// TIA Portal V20 export
FUNCTION_BLOCK "LER_Thickness"   // FB10, LAD
// stored: Access Published, MemoryReserve 100, SetENOAutomatically false
   VAR_INPUT
      enable : Bool := true;
      enableManualCmds : Bool;
      productUnused : Bool;   // Unused is simulation, dryrun etc..
      errAckHmi : Bool;
   END_VAR
   VAR_OUTPUT
      error : Bool;
      errorCode : Word;
   END_VAR
   VAR_IN_OUT
      configuration : "LER_typeThicknessConfiguration";
      moduleInterface : "LER_typeThicknessInterface";
      controlNodes : "LER_typeThicknessControlNode";
   END_VAR
   VAR
      statLVDTCmd { S7_SetPoint := 'True'} : "LER_typeThicknessCommand";
      statLVDTProfinetInput { S7_SetPoint := 'True'} : "LER_typeThicknessProfinetInput";
      statLVDTProfinetOutput { S7_SetPoint := 'True'} : "LER_typeThicknessProfinetOutput";
      statMonitoring : "LER_typeThicknessMonitoring";
      statLvdtConfig { S7_SetPoint := 'True'} : "LER_typeThicknessConfiguration";
      statRetValInt : Array[1..#count] of Int;
      statRetValWord { ExternalAccessible := 'False'; ExternalVisible := 'False'; ExternalWritable := 'False'} : Array[1..#count] of Word;
      instTON { S7_SetPoint := 'True'} : Array[0..4] of TON_TIME;
      statBit { S7_SetPoint := 'True'} : Array[0..49] of Bool;
      statRowDataDint_always : Array[0..3] of DInt;
      statRowDataReal_always : Array[0..3] of Real;
      statRowDataDint_capture : Array[0..3] of DInt;
      statRowDataReal_capture : Array[0..3] of Real;
      statTonTimer { S7_SetPoint := 'True'} : Array[0..99] of TON_TIME;
      statPulse { S7_SetPoint := 'True'} : Array[0..99] of Bool;
   END_VAR
   VAR_TEMP
      tempRetVal : Array[1..#count] of Int;
      tempIndex : Int;
   END_VAR
   VAR CONSTANT
      delayTime : Time := T#2s;
      count : Int := 10;
      scaleData : DInt := 256;
      scaleDigit : Real := 10000.0;
      statusNoErrorOccurred : Word := 16#0000;   // No error occurred.
      ioDeviceError : Word := 16#8000;
      ampError : Word := 16#8002;
      errHwdNotConfigured : Word := 16#8090;   // You have not configured a module for the specified hardware identifier or You have ignored the restriction concerning the length of consistent data, or you have not specified a hardware identifier as an address at parameter LADDR
      errRecordDataType : Word := 16#8092;   // Non-supported data type in the RECORD parameter.
      errNoDpProfinetIoModule : Word := 16#8093;   // No DP module/PROFINET IO device from which you can read consistent data exists for the hardware identifier specified in LADDR . This error code also occurs if the module addressed by means of LADDR does not have inputs.
      errIoAccessPermission : Word := 16#80A0;   // An access error was detected when accessing the I/O.
      errRecordLengthInsufficient : Word := 16#80B1;   // The length of the specified destination area at parameter RECORD is shorter than the configured user data length.
      errDataNotReceived : Word := 16#80C0;   // The data have not been read yet.
   END_VAR
   // // statBit[20] : amp0 OK
   // // statBit[21] : amp1 OK
   // // statBit[22] : amp2 OK
   // // statBit[23] : amp3 OK
   // // statBit[25] : Total OK
   // // statBit[30] : amp0 NG
   // // statBit[31] : amp1 NG
   // // statBit[32] : amp2 NG
   // // statBit[33] : amp3 NG
   // // statBit[35] : One or more NG
   // // statBit[40] : Busy
   // // statBit[41] : Complete
   // // statBit[45] : P_TRIG
   VAR_TEMP   // added for the SCL form of the ladder/FBD networks
      _w1 : Bool;
      _w2 : Bool;
      _w3 : Bool;
      _w4 : Bool;
      _w5 : Bool;
   END_VAR
BEGIN

REGION Network 1 (SCL): DP READ
   REGION DP read

       IF #enable AND NOT #productUnused THEN
           #statRetValInt[1] := DPRD_DAT(LADDR := #configuration.hwID.interfaceControllerID, RECORD => #statLVDTProfinetInput.interfaceController);
           #statRetValInt[2] := DPRD_DAT(LADDR := #configuration.hwID.ampID[0], RECORD => #statLVDTProfinetInput.amp[0]);
           #statRetValInt[3] := DPRD_DAT(LADDR := #configuration.hwID.ampID[1], RECORD => #statLVDTProfinetInput.amp[1]);
           #statRetValInt[4] := DPRD_DAT(LADDR := #configuration.hwID.ampID[2], RECORD => #statLVDTProfinetInput.amp[2]);
           #statRetValInt[5] := DPRD_DAT(LADDR := #configuration.hwID.ampID[3], RECORD => #statLVDTProfinetInput.amp[3]);
       END_IF;

   END_REGION
END_REGION

REGION Network 2 (SCL): INPUT MAPPING
   REGION Input mapping

       IF #enable THEN
           IF #enableManualCmds THEN
               #statLVDTCmd := #moduleInterface.command;
               #statLvdtConfig := #moduleInterface.configuration;
           ELSE
               #statLVDTCmd := #controlNodes.command;
               #statLvdtConfig := #configuration;
           END_IF;
       END_IF;

   END_REGION
END_REGION

REGION Network 3 (SCL): ERROR STATUS
   REGION Error check

       IF #enable AND NOT #productUnused THEN
           IF #statRetValInt <> #tempRetVal THEN
               FOR #tempIndex := 1 TO #count DO
                   #statRetValWord[#tempIndex] := INT_TO_WORD(#statRetValInt[#tempIndex]);
                   CASE #statRetValWord[#tempIndex] OF

                       #errHwdNotConfigured:
                           #errorCode := #errHwdNotConfigured;

                       #errRecordDataType:
                           #errorCode := #errRecordDataType;

                       #errNoDpProfinetIoModule:
                           #errorCode := #errNoDpProfinetIoModule;

                       #errIoAccessPermission:
                           #errorCode := #errIoAccessPermission;

                       #errRecordLengthInsufficient:
                           #errorCode := #errRecordLengthInsufficient;

                       #errDataNotReceived:
                           #errorCode := #errDataNotReceived;
                   END_CASE;
               END_FOR;

           ELSIF #statLVDTProfinetInput.interfaceController.b07ErrorStatus THEN
               #errorCode := #ioDeviceError;

           ELSIF #statLVDTProfinetInput.amp[0].b17ErrorStatus OR
               #statLVDTProfinetInput.amp[1].b17ErrorStatus OR
               #statLVDTProfinetInput.amp[2].b17ErrorStatus OR
               #statLVDTProfinetInput.amp[3].b17ErrorStatus THEN
               #errorCode := #ampError;

           ELSE
               #errorCode := #statusNoErrorOccurred;
           END_IF;
       ELSE
           #errorCode := #statusNoErrorOccurred;
       END_IF;

       #error := #errorCode <> 0;

   END_REGION
END_REGION

REGION Network 4: SEQUENCE : READY
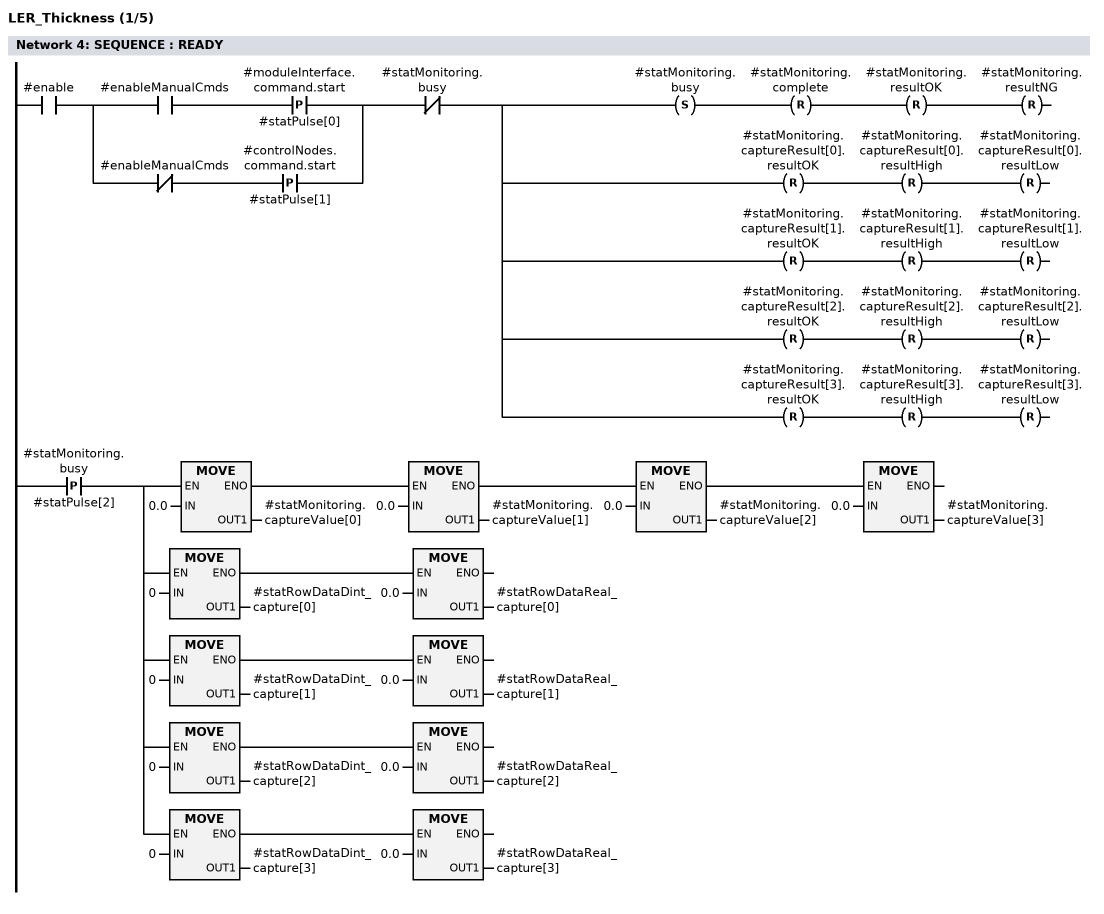
   RUNG wire#powerrail
      Contact( #enable )
      wire#w1
      Contact( #enableManualCmds )
      P_Contact(operand := #moduleInterface.command.start, bit := #statPulse[0])
      wire#w2
      I_Contact( #statMonitoring.busy )
      wire#w3
      S_Coil( #statMonitoring.busy )
      R_Coil( #statMonitoring.complete )
      R_Coil( #statMonitoring.resultOK )
      R_Coil( #statMonitoring.resultNG )
   END_RUNG
   RUNG wire#w1
      I_Contact( #enableManualCmds )
      P_Contact(operand := #controlNodes.command.start, bit := #statPulse[1])
   END_RUNG wire#w2
   RUNG wire#w3
      R_Coil( #statMonitoring.captureResult[0].resultOK )
      R_Coil( #statMonitoring.captureResult[0].resultHigh )
      R_Coil( #statMonitoring.captureResult[0].resultLow )
   END_RUNG
   RUNG wire#w3
      R_Coil( #statMonitoring.captureResult[1].resultOK )
      R_Coil( #statMonitoring.captureResult[1].resultHigh )
      R_Coil( #statMonitoring.captureResult[1].resultLow )
   END_RUNG
   RUNG wire#w3
      R_Coil( #statMonitoring.captureResult[2].resultOK )
      R_Coil( #statMonitoring.captureResult[2].resultHigh )
      R_Coil( #statMonitoring.captureResult[2].resultLow )
   END_RUNG
   RUNG wire#w3
      R_Coil( #statMonitoring.captureResult[3].resultOK )
      R_Coil( #statMonitoring.captureResult[3].resultHigh )
      R_Coil( #statMonitoring.captureResult[3].resultLow )
   END_RUNG
   RUNG wire#powerrail
      P_Contact(operand := #statMonitoring.busy, bit := #statPulse[2])
      wire#w4
      Move(in := 0.0, out1 => #statMonitoring.captureValue[0])
      Move(in := 0.0, out1 => #statMonitoring.captureValue[1])
      Move(in := 0.0, out1 => #statMonitoring.captureValue[2])
      Move(in := 0.0, out1 => #statMonitoring.captureValue[3])
   END_RUNG
   RUNG wire#w4
      Move(in := 0, out1 => #statRowDataDint_capture[0])
      Move(in := 0.0, out1 => #statRowDataReal_capture[0])
   END_RUNG
   RUNG wire#w4
      Move(in := 0, out1 => #statRowDataDint_capture[1])
      Move(in := 0.0, out1 => #statRowDataReal_capture[1])
   END_RUNG
   RUNG wire#w4
      Move(in := 0, out1 => #statRowDataDint_capture[2])
      Move(in := 0.0, out1 => #statRowDataReal_capture[2])
   END_RUNG
   RUNG wire#w4
      Move(in := 0, out1 => #statRowDataDint_capture[3])
      Move(in := 0.0, out1 => #statRowDataReal_capture[3])
   END_RUNG
   // the same network as SCL:
   #_w1 := #enable AND #enableManualCmds AND #moduleInterface.command.start AND NOT #statPulse[0];   // rising edge of #moduleInterface.command.start
   #statPulse[0] := #moduleInterface.command.start;
   #_w2 := #enable AND NOT #enableManualCmds AND #controlNodes.command.start AND NOT #statPulse[1];   // rising edge of #controlNodes.command.start
   #statPulse[1] := #controlNodes.command.start;
   #_w3 := (#_w1 OR #_w2) AND NOT #statMonitoring.busy;
   IF #_w3 THEN
       #statMonitoring.busy := TRUE;
       #statMonitoring.complete := FALSE;
       #statMonitoring.resultOK := FALSE;
       #statMonitoring.resultNG := FALSE;
       #statMonitoring.captureResult[0].resultOK := FALSE;
       #statMonitoring.captureResult[0].resultHigh := FALSE;
       #statMonitoring.captureResult[0].resultLow := FALSE;
       #statMonitoring.captureResult[1].resultOK := FALSE;
       #statMonitoring.captureResult[1].resultHigh := FALSE;
       #statMonitoring.captureResult[1].resultLow := FALSE;
       #statMonitoring.captureResult[2].resultOK := FALSE;
       #statMonitoring.captureResult[2].resultHigh := FALSE;
       #statMonitoring.captureResult[2].resultLow := FALSE;
       #statMonitoring.captureResult[3].resultOK := FALSE;
       #statMonitoring.captureResult[3].resultHigh := FALSE;
       #statMonitoring.captureResult[3].resultLow := FALSE;
   END_IF;
   #_w4 := #statMonitoring.busy AND NOT #statPulse[2];   // rising edge of #statMonitoring.busy
   #statPulse[2] := #statMonitoring.busy;
   IF #_w4 THEN
       #statMonitoring.captureValue[0] := 0.0;
       #statMonitoring.captureValue[1] := 0.0;
       #statMonitoring.captureValue[2] := 0.0;
       #statMonitoring.captureValue[3] := 0.0;
       #statRowDataDint_capture[0] := 0;
       #statRowDataReal_capture[0] := 0.0;
       #statRowDataDint_capture[1] := 0;
       #statRowDataReal_capture[1] := 0.0;
       #statRowDataDint_capture[2] := 0;
       #statRowDataReal_capture[2] := 0.0;
       #statRowDataDint_capture[3] := 0;
       #statRowDataReal_capture[3] := 0.0;
   END_IF;
END_REGION

REGION Network 5: SEQUENCE : START
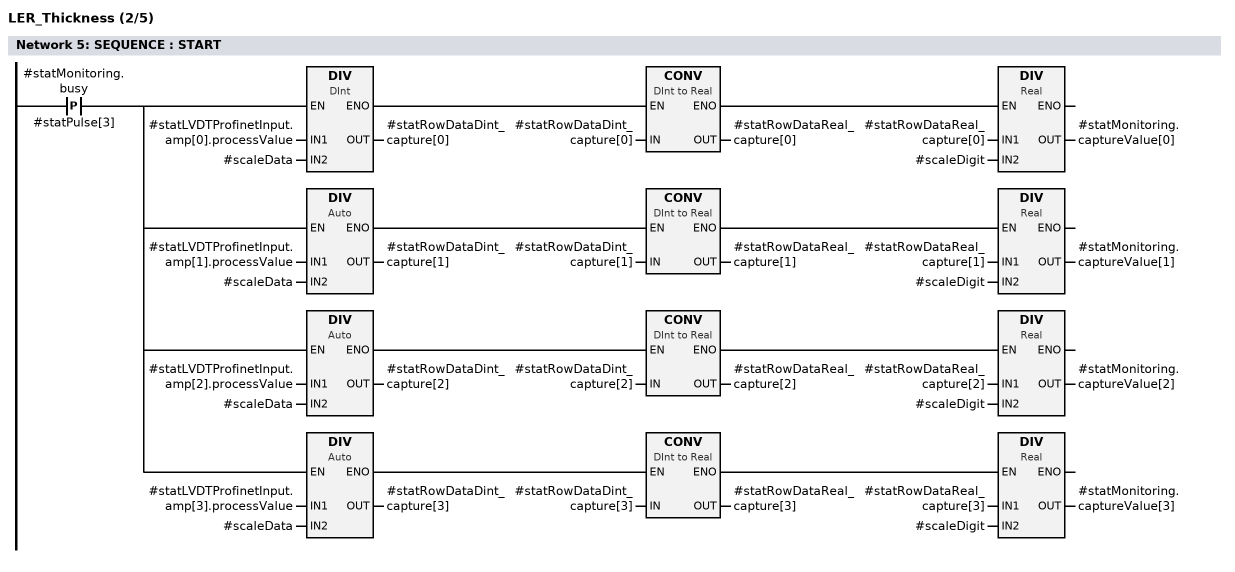
   RUNG wire#powerrail
      P_Contact(operand := #statMonitoring.busy, bit := #statPulse[3])
      wire#w1
      { S7_Templates := "SrcType := DInt" } Div(in1 := #statLVDTProfinetInput.amp[0].processValue, in2 := #scaleData, out => #statRowDataDint_capture[0])
      { S7_Templates := "[SrcType := DInt, DestType := Real]" } Convert(in := #statRowDataDint_capture[0], out => #statRowDataReal_capture[0])
      { S7_Templates := "SrcType := Real" } Div(in1 := #statRowDataReal_capture[0], in2 := #scaleDigit, out => #statMonitoring.captureValue[0])
   END_RUNG
   RUNG wire#w1
      Div(in1 := #statLVDTProfinetInput.amp[1].processValue, in2 := #scaleData, out => #statRowDataDint_capture[1])
      { S7_Templates := "[SrcType := DInt, DestType := Real]" } Convert(in := #statRowDataDint_capture[1], out => #statRowDataReal_capture[1])
      { S7_Templates := "SrcType := Real" } Div(in1 := #statRowDataReal_capture[1], in2 := #scaleDigit, out => #statMonitoring.captureValue[1])
   END_RUNG
   RUNG wire#w1
      Div(in1 := #statLVDTProfinetInput.amp[2].processValue, in2 := #scaleData, out => #statRowDataDint_capture[2])
      { S7_Templates := "[SrcType := DInt, DestType := Real]" } Convert(in := #statRowDataDint_capture[2], out => #statRowDataReal_capture[2])
      { S7_Templates := "SrcType := Real" } Div(in1 := #statRowDataReal_capture[2], in2 := #scaleDigit, out => #statMonitoring.captureValue[2])
   END_RUNG
   RUNG wire#w1
      Div(in1 := #statLVDTProfinetInput.amp[3].processValue, in2 := #scaleData, out => #statRowDataDint_capture[3])
      { S7_Templates := "[SrcType := DInt, DestType := Real]" } Convert(in := #statRowDataDint_capture[3], out => #statRowDataReal_capture[3])
      { S7_Templates := "SrcType := Real" } Div(in1 := #statRowDataReal_capture[3], in2 := #scaleDigit, out => #statMonitoring.captureValue[3])
   END_RUNG
   // the same network as SCL:
   #_w1 := #statMonitoring.busy AND NOT #statPulse[3];   // rising edge of #statMonitoring.busy
   #statPulse[3] := #statMonitoring.busy;
   IF #_w1 THEN
       #statRowDataDint_capture[0] := #statLVDTProfinetInput.amp[0].processValue / #scaleData;
       #statRowDataReal_capture[0] := DINT_TO_REAL(#statRowDataDint_capture[0]);
       #statMonitoring.captureValue[0] := #statRowDataReal_capture[0] / #scaleDigit;
       #statRowDataDint_capture[1] := #statLVDTProfinetInput.amp[1].processValue / #scaleData;
       #statRowDataReal_capture[1] := DINT_TO_REAL(#statRowDataDint_capture[1]);
       #statMonitoring.captureValue[1] := #statRowDataReal_capture[1] / #scaleDigit;
       #statRowDataDint_capture[2] := #statLVDTProfinetInput.amp[2].processValue / #scaleData;
       #statRowDataReal_capture[2] := DINT_TO_REAL(#statRowDataDint_capture[2]);
       #statMonitoring.captureValue[2] := #statRowDataReal_capture[2] / #scaleDigit;
       #statRowDataDint_capture[3] := #statLVDTProfinetInput.amp[3].processValue / #scaleData;
       #statRowDataReal_capture[3] := DINT_TO_REAL(#statRowDataDint_capture[3]);
       #statMonitoring.captureValue[3] := #statRowDataReal_capture[3] / #scaleDigit;
   END_IF;
END_REGION

REGION Network 6: SEQUENCE : RESULT
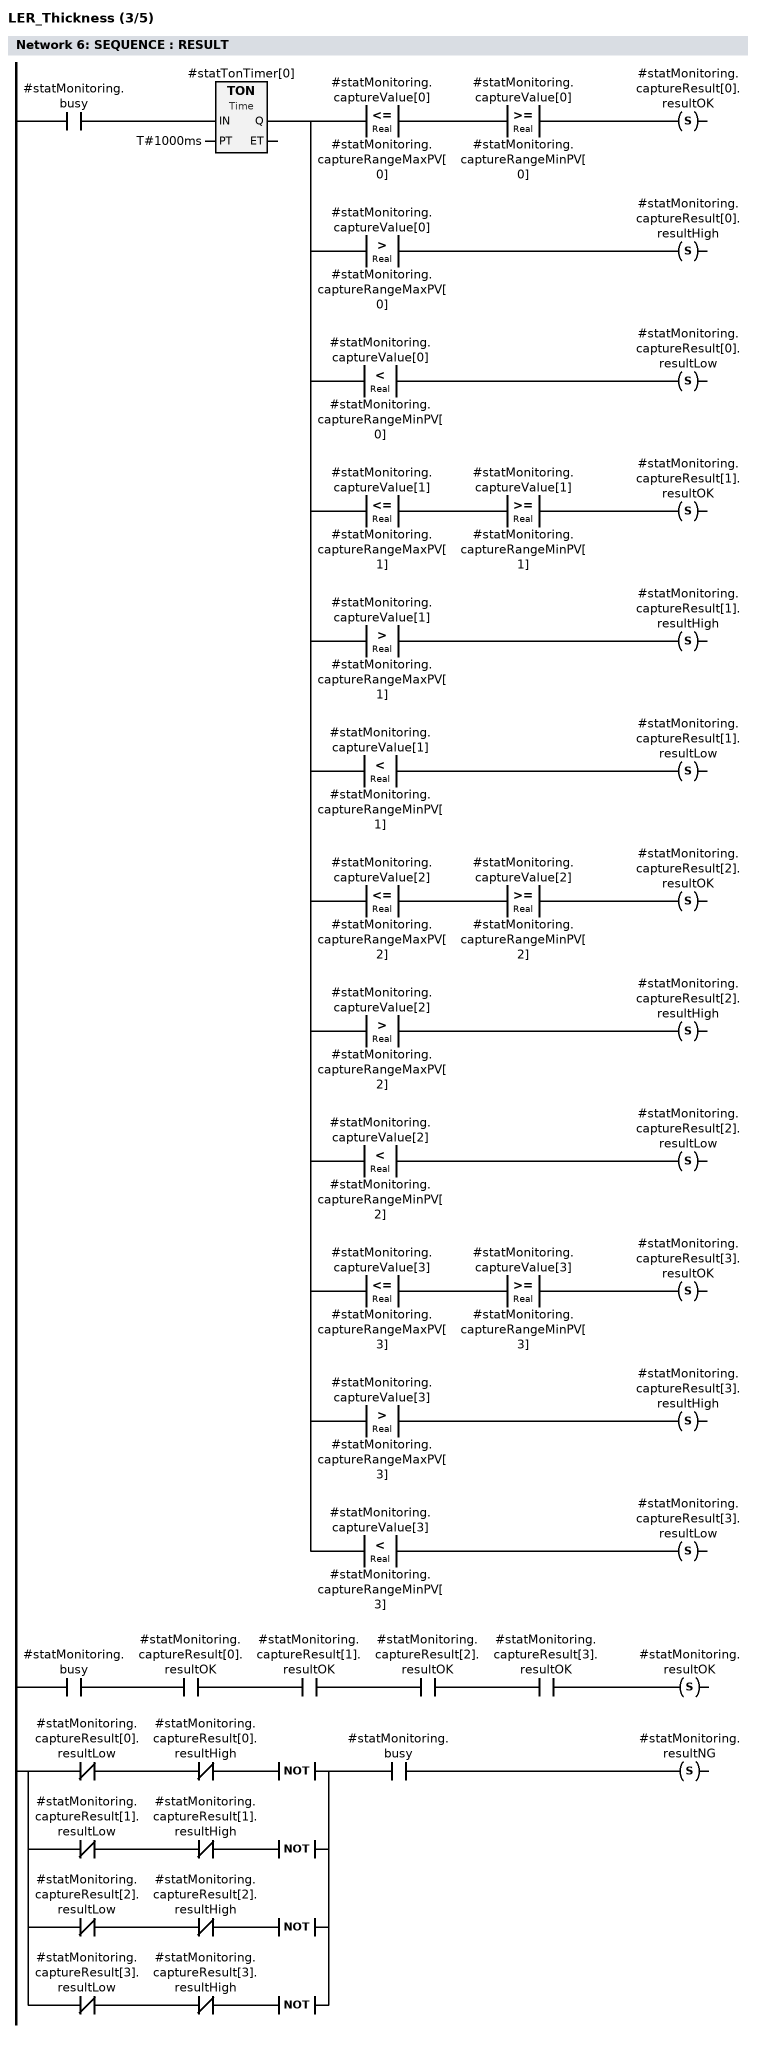
   RUNG wire#powerrail
      Contact( #statMonitoring.busy )
      { S7_Templates := "time_type := Time" } #statTonTimer[0].TON(pt := T#1000ms, et =>)
      wire#w1
      { S7_Templates := "SrcType := Real" } LE_Contact(in1 := #statMonitoring.captureValue[0], in2 := #statMonitoring.captureRangeMaxPV[0])
      { S7_Templates := "SrcType := Real" } GE_Contact(in1 := #statMonitoring.captureValue[0], in2 := #statMonitoring.captureRangeMinPV[0])
      S_Coil( #statMonitoring.captureResult[0].resultOK )
   END_RUNG
   RUNG wire#w1
      { S7_Templates := "SrcType := Real" } GT_Contact(in1 := #statMonitoring.captureValue[0], in2 := #statMonitoring.captureRangeMaxPV[0])
      S_Coil( #statMonitoring.captureResult[0].resultHigh )
   END_RUNG
   RUNG wire#w1
      { S7_Templates := "SrcType := Real" } LT_Contact(in1 := #statMonitoring.captureValue[0], in2 := #statMonitoring.captureRangeMinPV[0])
      S_Coil( #statMonitoring.captureResult[0].resultLow )
   END_RUNG
   RUNG wire#w1
      { S7_Templates := "SrcType := Real" } LE_Contact(in1 := #statMonitoring.captureValue[1], in2 := #statMonitoring.captureRangeMaxPV[1])
      { S7_Templates := "SrcType := Real" } GE_Contact(in1 := #statMonitoring.captureValue[1], in2 := #statMonitoring.captureRangeMinPV[1])
      S_Coil( #statMonitoring.captureResult[1].resultOK )
   END_RUNG
   RUNG wire#w1
      { S7_Templates := "SrcType := Real" } GT_Contact(in1 := #statMonitoring.captureValue[1], in2 := #statMonitoring.captureRangeMaxPV[1])
      S_Coil( #statMonitoring.captureResult[1].resultHigh )
   END_RUNG
   RUNG wire#w1
      { S7_Templates := "SrcType := Real" } LT_Contact(in1 := #statMonitoring.captureValue[1], in2 := #statMonitoring.captureRangeMinPV[1])
      S_Coil( #statMonitoring.captureResult[1].resultLow )
   END_RUNG
   RUNG wire#w1
      { S7_Templates := "SrcType := Real" } LE_Contact(in1 := #statMonitoring.captureValue[2], in2 := #statMonitoring.captureRangeMaxPV[2])
      { S7_Templates := "SrcType := Real" } GE_Contact(in1 := #statMonitoring.captureValue[2], in2 := #statMonitoring.captureRangeMinPV[2])
      S_Coil( #statMonitoring.captureResult[2].resultOK )
   END_RUNG
   RUNG wire#w1
      { S7_Templates := "SrcType := Real" } GT_Contact(in1 := #statMonitoring.captureValue[2], in2 := #statMonitoring.captureRangeMaxPV[2])
      S_Coil( #statMonitoring.captureResult[2].resultHigh )
   END_RUNG
   RUNG wire#w1
      { S7_Templates := "SrcType := Real" } LT_Contact(in1 := #statMonitoring.captureValue[2], in2 := #statMonitoring.captureRangeMinPV[2])
      S_Coil( #statMonitoring.captureResult[2].resultLow )
   END_RUNG
   RUNG wire#w1
      { S7_Templates := "SrcType := Real" } LE_Contact(in1 := #statMonitoring.captureValue[3], in2 := #statMonitoring.captureRangeMaxPV[3])
      { S7_Templates := "SrcType := Real" } GE_Contact(in1 := #statMonitoring.captureValue[3], in2 := #statMonitoring.captureRangeMinPV[3])
      S_Coil( #statMonitoring.captureResult[3].resultOK )
   END_RUNG
   RUNG wire#w1
      { S7_Templates := "SrcType := Real" } GT_Contact(in1 := #statMonitoring.captureValue[3], in2 := #statMonitoring.captureRangeMaxPV[3])
      S_Coil( #statMonitoring.captureResult[3].resultHigh )
   END_RUNG
   RUNG wire#w1
      { S7_Templates := "SrcType := Real" } LT_Contact(in1 := #statMonitoring.captureValue[3], in2 := #statMonitoring.captureRangeMinPV[3])
      S_Coil( #statMonitoring.captureResult[3].resultLow )
   END_RUNG
   RUNG wire#powerrail
      Contact( #statMonitoring.busy )
      Contact( #statMonitoring.captureResult[0].resultOK )
      Contact( #statMonitoring.captureResult[1].resultOK )
      Contact( #statMonitoring.captureResult[2].resultOK )
      Contact( #statMonitoring.captureResult[3].resultOK )
      S_Coil( #statMonitoring.resultOK )
   END_RUNG
   RUNG wire#powerrail
      I_Contact( #statMonitoring.captureResult[0].resultLow )
      I_Contact( #statMonitoring.captureResult[0].resultHigh )
      Not()
      wire#w2
      Contact( #statMonitoring.busy )
      S_Coil( #statMonitoring.resultNG )
   END_RUNG
   RUNG wire#powerrail
      I_Contact( #statMonitoring.captureResult[1].resultLow )
      I_Contact( #statMonitoring.captureResult[1].resultHigh )
      Not()
   END_RUNG wire#w2
   RUNG wire#powerrail
      I_Contact( #statMonitoring.captureResult[2].resultLow )
      I_Contact( #statMonitoring.captureResult[2].resultHigh )
      Not()
   END_RUNG wire#w2
   RUNG wire#powerrail
      I_Contact( #statMonitoring.captureResult[3].resultLow )
      I_Contact( #statMonitoring.captureResult[3].resultHigh )
      Not()
   END_RUNG wire#w2
   // the same network as SCL:
   #statTonTimer[0].TON(IN := #statMonitoring.busy, PT := T#1000ms);
   IF #statTonTimer[0].Q AND (#statMonitoring.captureValue[0] <= #statMonitoring.captureRangeMaxPV[0]) AND (#statMonitoring.captureValue[0] >= #statMonitoring.captureRangeMinPV[0]) THEN
       #statMonitoring.captureResult[0].resultOK := TRUE;
   END_IF;
   IF #statTonTimer[0].Q AND (#statMonitoring.captureValue[0] > #statMonitoring.captureRangeMaxPV[0]) THEN
       #statMonitoring.captureResult[0].resultHigh := TRUE;
   END_IF;
   IF #statTonTimer[0].Q AND (#statMonitoring.captureValue[0] < #statMonitoring.captureRangeMinPV[0]) THEN
       #statMonitoring.captureResult[0].resultLow := TRUE;
   END_IF;
   IF #statTonTimer[0].Q AND (#statMonitoring.captureValue[1] <= #statMonitoring.captureRangeMaxPV[1]) AND (#statMonitoring.captureValue[1] >= #statMonitoring.captureRangeMinPV[1]) THEN
       #statMonitoring.captureResult[1].resultOK := TRUE;
   END_IF;
   IF #statTonTimer[0].Q AND (#statMonitoring.captureValue[1] > #statMonitoring.captureRangeMaxPV[1]) THEN
       #statMonitoring.captureResult[1].resultHigh := TRUE;
   END_IF;
   IF #statTonTimer[0].Q AND (#statMonitoring.captureValue[1] < #statMonitoring.captureRangeMinPV[1]) THEN
       #statMonitoring.captureResult[1].resultLow := TRUE;
   END_IF;
   IF #statTonTimer[0].Q AND (#statMonitoring.captureValue[2] <= #statMonitoring.captureRangeMaxPV[2]) AND (#statMonitoring.captureValue[2] >= #statMonitoring.captureRangeMinPV[2]) THEN
       #statMonitoring.captureResult[2].resultOK := TRUE;
   END_IF;
   IF #statTonTimer[0].Q AND (#statMonitoring.captureValue[2] > #statMonitoring.captureRangeMaxPV[2]) THEN
       #statMonitoring.captureResult[2].resultHigh := TRUE;
   END_IF;
   IF #statTonTimer[0].Q AND (#statMonitoring.captureValue[2] < #statMonitoring.captureRangeMinPV[2]) THEN
       #statMonitoring.captureResult[2].resultLow := TRUE;
   END_IF;
   IF #statTonTimer[0].Q AND (#statMonitoring.captureValue[3] <= #statMonitoring.captureRangeMaxPV[3]) AND (#statMonitoring.captureValue[3] >= #statMonitoring.captureRangeMinPV[3]) THEN
       #statMonitoring.captureResult[3].resultOK := TRUE;
   END_IF;
   IF #statTonTimer[0].Q AND (#statMonitoring.captureValue[3] > #statMonitoring.captureRangeMaxPV[3]) THEN
       #statMonitoring.captureResult[3].resultHigh := TRUE;
   END_IF;
   IF #statTonTimer[0].Q AND (#statMonitoring.captureValue[3] < #statMonitoring.captureRangeMinPV[3]) THEN
       #statMonitoring.captureResult[3].resultLow := TRUE;
   END_IF;
   IF #statMonitoring.busy AND #statMonitoring.captureResult[0].resultOK AND #statMonitoring.captureResult[1].resultOK AND #statMonitoring.captureResult[2].resultOK AND #statMonitoring.captureResult[3].resultOK THEN
       #statMonitoring.resultOK := TRUE;
   END_IF;
   IF (NOT (NOT #statMonitoring.captureResult[0].resultLow AND NOT #statMonitoring.captureResult[0].resultHigh) OR NOT (NOT #statMonitoring.captureResult[1].resultLow AND NOT #statMonitoring.captureResult[1].resultHigh) OR NOT (NOT #statMonitoring.captureResult[2].resultLow AND NOT #statMonitoring.captureResult[2].resultHigh) OR NOT (NOT #statMonitoring.captureResult[3].resultLow AND NOT #statMonitoring.captureResult[3].resultHigh)) AND #statMonitoring.busy THEN
       #statMonitoring.resultNG := TRUE;
   END_IF;
END_REGION

REGION Network 7: SEQUENCE : COMPLETE
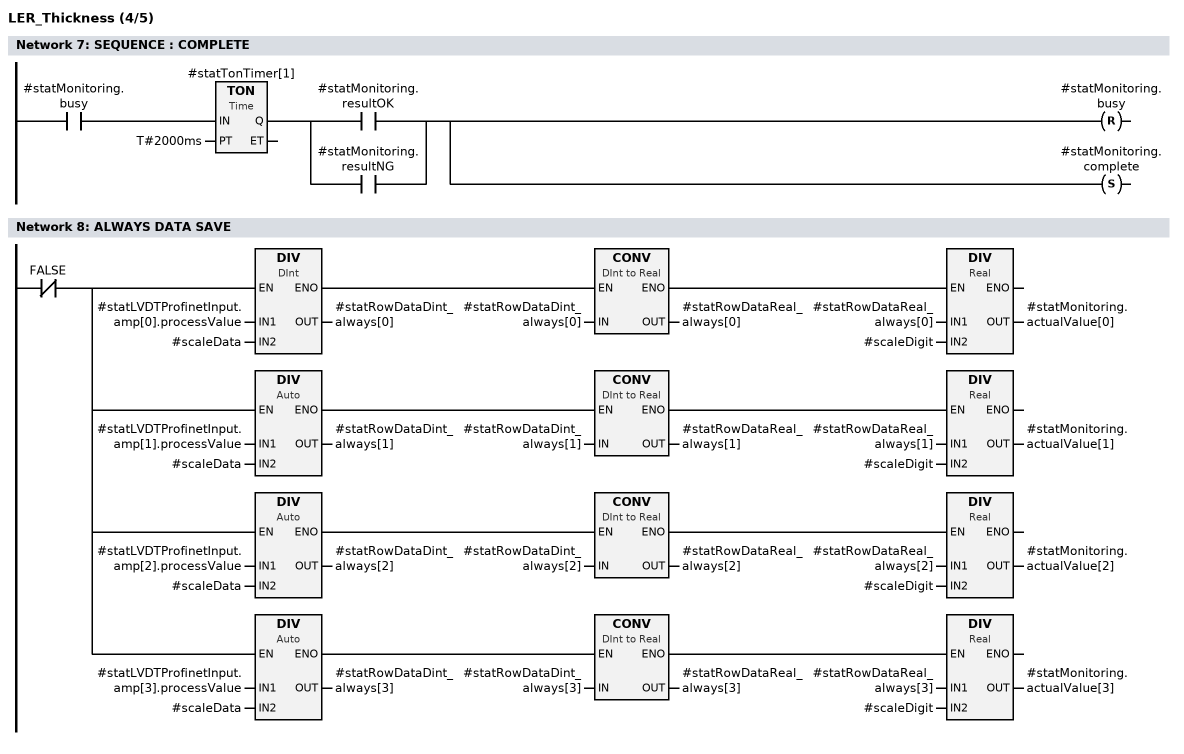
   RUNG wire#powerrail
      Contact( #statMonitoring.busy )
      { S7_Templates := "time_type := Time" } #statTonTimer[1].TON(pt := T#2000ms, et =>)
      wire#w1
      Contact( #statMonitoring.resultOK )
      wire#w2
      R_Coil( #statMonitoring.busy )
   END_RUNG
   RUNG wire#w1
      Contact( #statMonitoring.resultNG )
   END_RUNG wire#w2
   RUNG wire#w2
      S_Coil( #statMonitoring.complete )
   END_RUNG
   // the same network as SCL:
   #statTonTimer[1].TON(IN := #statMonitoring.busy, PT := T#2000ms);
   IF #statTonTimer[1].Q AND (#statMonitoring.resultOK OR #statMonitoring.resultNG) THEN
       #statMonitoring.busy := FALSE;
       #statMonitoring.complete := TRUE;
   END_IF;
END_REGION

REGION Network 8: ALWAYS DATA SAVE
   RUNG wire#powerrail
      I_Contact( FALSE )
      wire#w1
      { S7_Templates := "SrcType := DInt" } Div(in1 := #statLVDTProfinetInput.amp[0].processValue, in2 := #scaleData, out => #statRowDataDint_always[0])
      { S7_Templates := "[SrcType := DInt, DestType := Real]" } Convert(in := #statRowDataDint_always[0], out => #statRowDataReal_always[0])
      { S7_Templates := "SrcType := Real" } Div(in1 := #statRowDataReal_always[0], in2 := #scaleDigit, out => #statMonitoring.actualValue[0])
   END_RUNG
   RUNG wire#w1
      Div(in1 := #statLVDTProfinetInput.amp[1].processValue, in2 := #scaleData, out => #statRowDataDint_always[1])
      { S7_Templates := "[SrcType := DInt, DestType := Real]" } Convert(in := #statRowDataDint_always[1], out => #statRowDataReal_always[1])
      { S7_Templates := "SrcType := Real" } Div(in1 := #statRowDataReal_always[1], in2 := #scaleDigit, out => #statMonitoring.actualValue[1])
   END_RUNG
   RUNG wire#w1
      Div(in1 := #statLVDTProfinetInput.amp[2].processValue, in2 := #scaleData, out => #statRowDataDint_always[2])
      { S7_Templates := "[SrcType := DInt, DestType := Real]" } Convert(in := #statRowDataDint_always[2], out => #statRowDataReal_always[2])
      { S7_Templates := "SrcType := Real" } Div(in1 := #statRowDataReal_always[2], in2 := #scaleDigit, out => #statMonitoring.actualValue[2])
   END_RUNG
   RUNG wire#w1
      Div(in1 := #statLVDTProfinetInput.amp[3].processValue, in2 := #scaleData, out => #statRowDataDint_always[3])
      { S7_Templates := "[SrcType := DInt, DestType := Real]" } Convert(in := #statRowDataDint_always[3], out => #statRowDataReal_always[3])
      { S7_Templates := "SrcType := Real" } Div(in1 := #statRowDataReal_always[3], in2 := #scaleDigit, out => #statMonitoring.actualValue[3])
   END_RUNG
   // the same network as SCL:
   IF NOT FALSE THEN
       #statRowDataDint_always[0] := #statLVDTProfinetInput.amp[0].processValue / #scaleData;
       #statRowDataReal_always[0] := DINT_TO_REAL(#statRowDataDint_always[0]);
       #statMonitoring.actualValue[0] := #statRowDataReal_always[0] / #scaleDigit;
       #statRowDataDint_always[1] := #statLVDTProfinetInput.amp[1].processValue / #scaleData;
       #statRowDataReal_always[1] := DINT_TO_REAL(#statRowDataDint_always[1]);
       #statMonitoring.actualValue[1] := #statRowDataReal_always[1] / #scaleDigit;
       #statRowDataDint_always[2] := #statLVDTProfinetInput.amp[2].processValue / #scaleData;
       #statRowDataReal_always[2] := DINT_TO_REAL(#statRowDataDint_always[2]);
       #statMonitoring.actualValue[2] := #statRowDataReal_always[2] / #scaleDigit;
       #statRowDataDint_always[3] := #statLVDTProfinetInput.amp[3].processValue / #scaleData;
       #statRowDataReal_always[3] := DINT_TO_REAL(#statRowDataDint_always[3]);
       #statMonitoring.actualValue[3] := #statRowDataReal_always[3] / #scaleDigit;
   END_IF;
END_REGION

REGION Network 9: ZERO SET
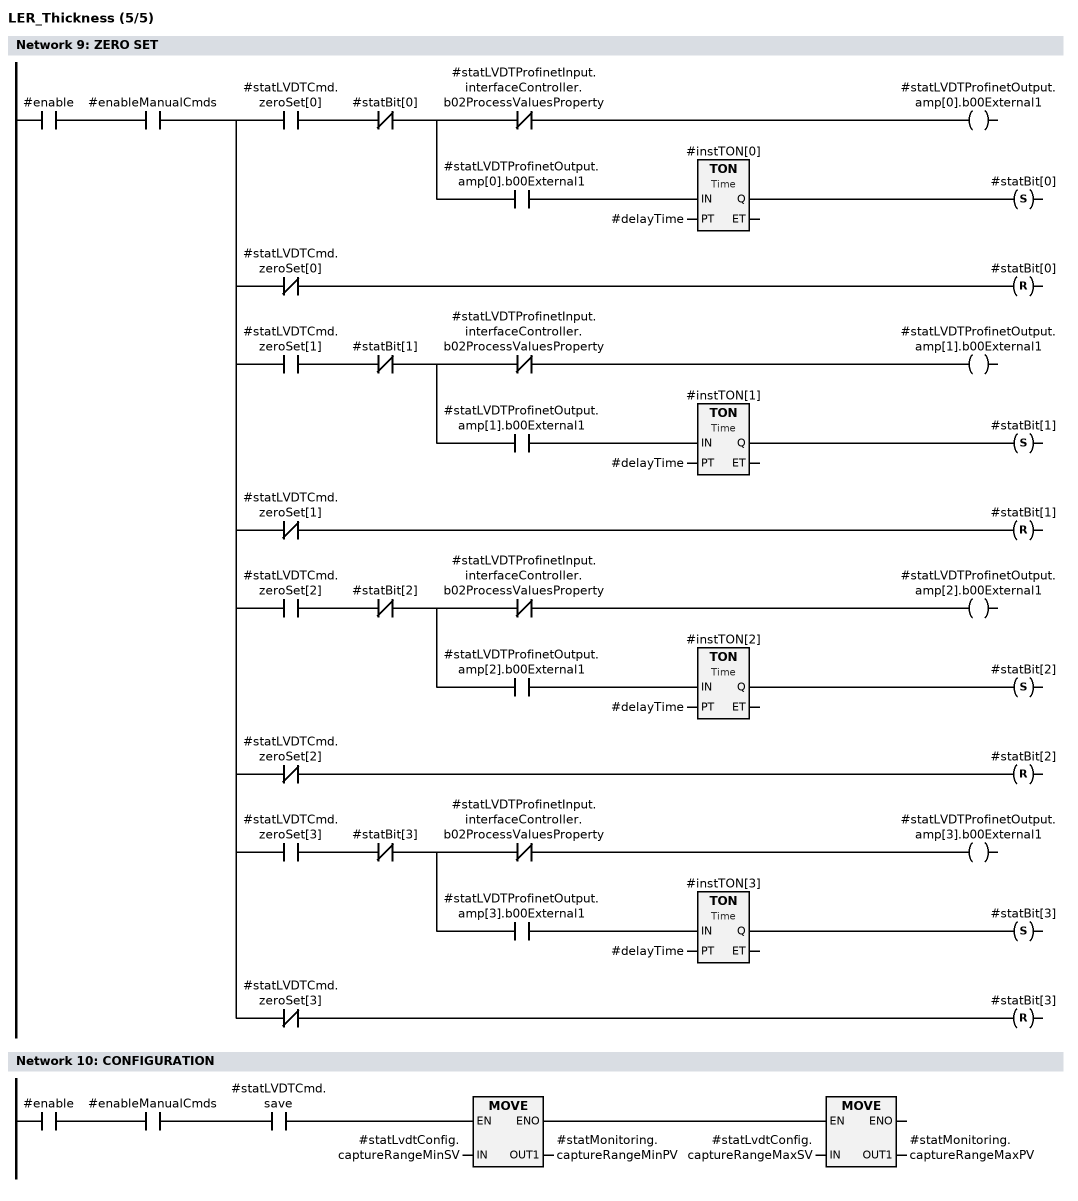
   RUNG wire#powerrail
      Contact( #enable )
      Contact( #enableManualCmds )
      wire#w1
      Contact( #statLVDTCmd.zeroSet[0] )
      I_Contact( #statBit[0] )
      wire#w2
      I_Contact( #statLVDTProfinetInput.interfaceController.b02ProcessValuesProperty )
      Coil( #statLVDTProfinetOutput.amp[0].b00External1 )
   END_RUNG
   RUNG wire#w2
      Contact( #statLVDTProfinetOutput.amp[0].b00External1 )
      { S7_Templates := "time_type := Time" } #instTON[0].TON(pt := #delayTime, et =>)
      S_Coil( #statBit[0] )
   END_RUNG
   RUNG wire#w1
      I_Contact( #statLVDTCmd.zeroSet[0] )
      R_Coil( #statBit[0] )
   END_RUNG
   RUNG wire#w1
      Contact( #statLVDTCmd.zeroSet[1] )
      I_Contact( #statBit[1] )
      wire#w3
      I_Contact( #statLVDTProfinetInput.interfaceController.b02ProcessValuesProperty )
      Coil( #statLVDTProfinetOutput.amp[1].b00External1 )
   END_RUNG
   RUNG wire#w3
      Contact( #statLVDTProfinetOutput.amp[1].b00External1 )
      { S7_Templates := "time_type := Time" } #instTON[1].TON(pt := #delayTime, et =>)
      S_Coil( #statBit[1] )
   END_RUNG
   RUNG wire#w1
      I_Contact( #statLVDTCmd.zeroSet[1] )
      R_Coil( #statBit[1] )
   END_RUNG
   RUNG wire#w1
      Contact( #statLVDTCmd.zeroSet[2] )
      I_Contact( #statBit[2] )
      wire#w4
      I_Contact( #statLVDTProfinetInput.interfaceController.b02ProcessValuesProperty )
      Coil( #statLVDTProfinetOutput.amp[2].b00External1 )
   END_RUNG
   RUNG wire#w4
      Contact( #statLVDTProfinetOutput.amp[2].b00External1 )
      { S7_Templates := "time_type := Time" } #instTON[2].TON(pt := #delayTime, et =>)
      S_Coil( #statBit[2] )
   END_RUNG
   RUNG wire#w1
      I_Contact( #statLVDTCmd.zeroSet[2] )
      R_Coil( #statBit[2] )
   END_RUNG
   RUNG wire#w1
      Contact( #statLVDTCmd.zeroSet[3] )
      I_Contact( #statBit[3] )
      wire#w5
      I_Contact( #statLVDTProfinetInput.interfaceController.b02ProcessValuesProperty )
      Coil( #statLVDTProfinetOutput.amp[3].b00External1 )
   END_RUNG
   RUNG wire#w5
      Contact( #statLVDTProfinetOutput.amp[3].b00External1 )
      { S7_Templates := "time_type := Time" } #instTON[3].TON(pt := #delayTime, et =>)
      S_Coil( #statBit[3] )
   END_RUNG
   RUNG wire#w1
      I_Contact( #statLVDTCmd.zeroSet[3] )
      R_Coil( #statBit[3] )
   END_RUNG
   // the same network as SCL:
   #_w1 := #enable AND #enableManualCmds;
   #_w2 := #_w1 AND #statLVDTCmd.zeroSet[0] AND NOT #statBit[0];
   #statLVDTProfinetOutput.amp[0].b00External1 := #_w2 AND NOT #statLVDTProfinetInput.interfaceController.b02ProcessValuesProperty;
   #instTON[0].TON(IN := #_w2 AND #statLVDTProfinetOutput.amp[0].b00External1, PT := #delayTime);
   IF #instTON[0].Q THEN #statBit[0] := TRUE; END_IF;
   IF #_w1 AND NOT #statLVDTCmd.zeroSet[0] THEN #statBit[0] := FALSE; END_IF;
   #_w3 := #_w1 AND #statLVDTCmd.zeroSet[1] AND NOT #statBit[1];
   #statLVDTProfinetOutput.amp[1].b00External1 := #_w3 AND NOT #statLVDTProfinetInput.interfaceController.b02ProcessValuesProperty;
   #instTON[1].TON(IN := #_w3 AND #statLVDTProfinetOutput.amp[1].b00External1, PT := #delayTime);
   IF #instTON[1].Q THEN #statBit[1] := TRUE; END_IF;
   IF #_w1 AND NOT #statLVDTCmd.zeroSet[1] THEN #statBit[1] := FALSE; END_IF;
   #_w4 := #_w1 AND #statLVDTCmd.zeroSet[2] AND NOT #statBit[2];
   #statLVDTProfinetOutput.amp[2].b00External1 := #_w4 AND NOT #statLVDTProfinetInput.interfaceController.b02ProcessValuesProperty;
   #instTON[2].TON(IN := #_w4 AND #statLVDTProfinetOutput.amp[2].b00External1, PT := #delayTime);
   IF #instTON[2].Q THEN #statBit[2] := TRUE; END_IF;
   IF #_w1 AND NOT #statLVDTCmd.zeroSet[2] THEN #statBit[2] := FALSE; END_IF;
   #_w5 := #_w1 AND #statLVDTCmd.zeroSet[3] AND NOT #statBit[3];
   #statLVDTProfinetOutput.amp[3].b00External1 := #_w5 AND NOT #statLVDTProfinetInput.interfaceController.b02ProcessValuesProperty;
   #instTON[3].TON(IN := #_w5 AND #statLVDTProfinetOutput.amp[3].b00External1, PT := #delayTime);
   IF #instTON[3].Q THEN #statBit[3] := TRUE; END_IF;
   IF #_w1 AND NOT #statLVDTCmd.zeroSet[3] THEN #statBit[3] := FALSE; END_IF;
END_REGION

REGION Network 10: CONFIGURATION
   RUNG wire#powerrail
      Contact( #enable )
      Contact( #enableManualCmds )
      Contact( #statLVDTCmd.save )
      Move(in := #statLvdtConfig.captureRangeMinSV, out1 => #statMonitoring.captureRangeMinPV)
      Move(in := #statLvdtConfig.captureRangeMaxSV, out1 => #statMonitoring.captureRangeMaxPV)
   END_RUNG
   // the same network as SCL:
   IF #enable AND #enableManualCmds AND #statLVDTCmd.save THEN
       #statMonitoring.captureRangeMinPV := #statLvdtConfig.captureRangeMinSV;
       #statMonitoring.captureRangeMaxPV := #statLvdtConfig.captureRangeMaxSV;
   END_IF;
END_REGION

REGION Network 11 (SCL): DP WRITE
   REGION DP write

       #statRetValInt[6] := DPWR_DAT(LADDR := #configuration.hwID.interfaceControllerID, RECORD := #statLVDTProfinetOutput.interfaceController);
       #statRetValInt[7] := DPWR_DAT(LADDR := #configuration.hwID.ampID[0], RECORD := #statLVDTProfinetOutput.amp[0]);
       #statRetValInt[8] := DPWR_DAT(LADDR := #configuration.hwID.ampID[1], RECORD := #statLVDTProfinetOutput.amp[1]);
       #statRetValInt[9] := DPWR_DAT(LADDR := #configuration.hwID.ampID[2], RECORD := #statLVDTProfinetOutput.amp[2]);
       #statRetValInt[10] := DPWR_DAT(LADDR := #configuration.hwID.ampID[3], RECORD := #statLVDTProfinetOutput.amp[3]);

   END_REGION
END_REGION

REGION Network 12 (SCL): OUTPUT MAPPING
   REGION Output mapping

       #controlNodes.monitoring := #moduleInterface.monitoring := #statMonitoring;

   END_REGION
END_REGION
END_FUNCTION_BLOCK
